{attribute 'OPC.UA.DA.StructuredType' := '1'}
TYPE ST_AmbientState :
STRUCT
	fOutsideTemperature : REAL;
	fOutsideTemperature_Container : REAL;
	fOutsideTemperature_Mean : REAL;
	fHallTemperature : REAL;
	fRoomTemperature_Container : REAL;
	fWindSpeed : REAL;
	fDawn : REAL;
	bRain : BOOL;
	sTemperatureUnit : STRING := 'degreeC';
	sDawnUnit : STRING := 'lux';
	sWindSpeedUnit : STRING := 'm/s';
	fTemperatureSeminarRoom : REAL; //degreeC
	fCO2SeminarRoom 		: REAL; //Measured CO2 connection in ppm
	fTemperatureStudentRoom : REAL; //degreeC
	fCO2StudentRoom 		: REAL; //Measured CO2 connection in ppm
END_STRUCT
END_TYPE

(* stored: Version 1.1.0.1, ProductVersion 3.1.4024.10
   DUT ST_AmbientState: Id {18024053-1db6-499b-af8a-99fd20169e28} *)
